// TIA Portal project "Pozitif KT ile Basma Sayan Uygulaması" (V18)

(* hardware
DEVICE "S7-1200 station_1"  S7-1200 Station
   slot 0: "Rack_0"  S7-1200 Rack  Rack  V1.0
   slot 1: "PLC_1"  CPU 1214C AC/DC/Rly  6ES7 214-1BG40-0XB0  V4.6
*)

// ===== PLC "PLC_1"  CPU 1214C AC/DC/Rly =====

VAR_GLOBAL   // PLC tag table "Default tag table"
   "Stop" AT %I0.0 : Bool;
   "PKT" AT %I0.1 : Bool;
   "NKT" AT %I0.2 : Bool;
   "PKT_Yardımcı" AT %M0.0 : Bool;
   "Motor_1" AT %Q0.0 : Bool;
   "NKT_Yardımcı" AT %M0.1 : Bool;
   "Motor_2" AT %Q0.1 : Bool;
END_VAR

ORGANIZATION_BLOCK "Main"   // OB1, LAD, ProgramCycle
TITLE = "Main Program Sweep (Cycle)"
{ S7_Optimized_Access := 'TRUE' }
VERSION : 0.1
// Bir motorun kenar tetikleme ve set-reset komutlarını kullanarak çalıştırılıp durdurulmasını sağlamak.
   VAR_INPUT
      Initial_Call : Bool;   // Initial call of this OB
      Remanence : Bool;   // =True, if remanent data are available
   END_VAR
   VAR_TEMP   // added for the SCL form of the ladder/FBD networks
      _w1 : Bool;
   END_VAR
BEGIN

REGION Network 1
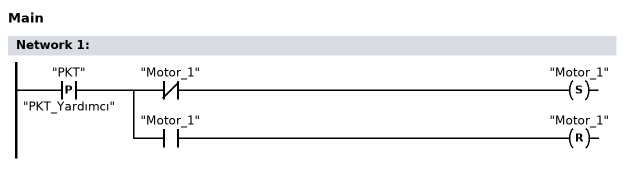
   RUNG wire#powerrail
      P_Contact(operand := "PKT", bit := "PKT_Yardımcı")
      wire#w1
      I_Contact( "Motor_1" )
      S_Coil( "Motor_1" )
   END_RUNG
   RUNG wire#w1
      Contact( "Motor_1" )
      R_Coil( "Motor_1" )
   END_RUNG
   // the same network as SCL:
   #_w1 := "PKT" AND NOT "PKT_Yardımcı";   // rising edge of "PKT"
   "PKT_Yardımcı" := "PKT";
   IF #_w1 AND NOT "Motor_1" THEN "Motor_1" := TRUE; END_IF;
   IF #_w1 AND "Motor_1" THEN "Motor_1" := FALSE; END_IF;
END_REGION
END_ORGANIZATION_BLOCK